// TIA Portal V20 export
FUNCTION "CallCycleTimer" : Void   // FC18, LAD
// stored: SetENOAutomatically false
   VAR CONSTANT
      TRUE : Bool := TRUE;
   END_VAR
BEGIN

REGION Network 1: Cycle Timer Em 0
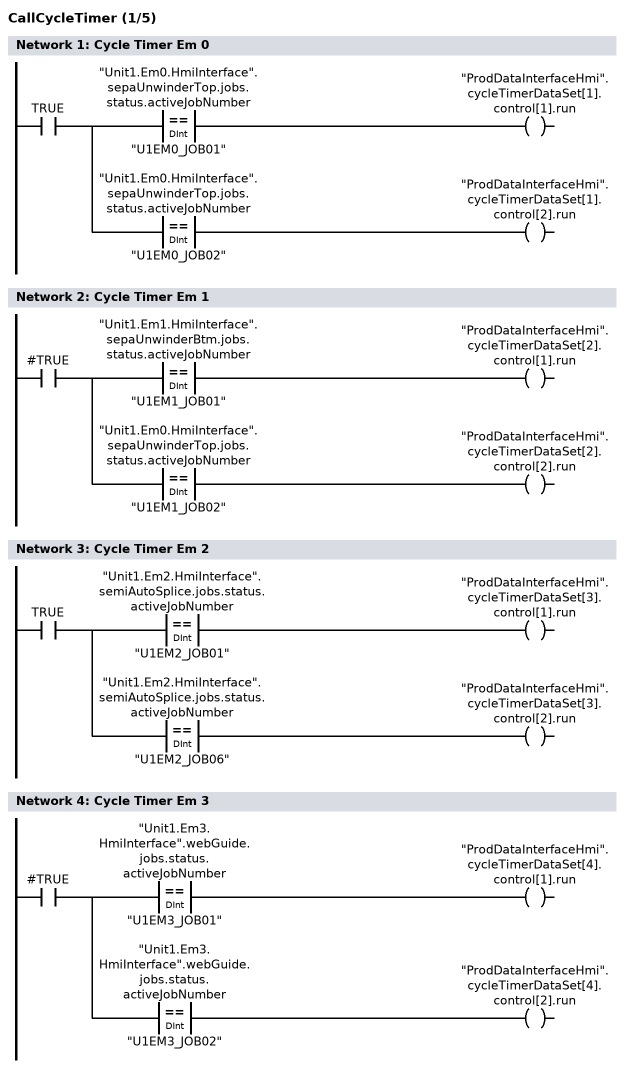
   RUNG wire#powerrail
      Contact( TRUE )
      wire#w1
      { S7_Templates := "SrcType := DInt" } EQ_Contact(in1 := "Unit1.Em0.HmiInterface".sepaUnwinderTop.jobs.status.activeJobNumber, in2 := "U1EM0_JOB01")
      Coil( "ProdDataInterfaceHmi".cycleTimerDataSet[1].control[1].run )
   END_RUNG
   RUNG wire#w1
      { S7_Templates := "SrcType := DInt" } EQ_Contact(in1 := "Unit1.Em0.HmiInterface".sepaUnwinderTop.jobs.status.activeJobNumber, in2 := "U1EM0_JOB02")
      Coil( "ProdDataInterfaceHmi".cycleTimerDataSet[1].control[2].run )
   END_RUNG
   // the same network as SCL:
   "ProdDataInterfaceHmi".cycleTimerDataSet[1].control[1].run := TRUE AND ("Unit1.Em0.HmiInterface".sepaUnwinderTop.jobs.status.activeJobNumber = "U1EM0_JOB01");
   "ProdDataInterfaceHmi".cycleTimerDataSet[1].control[2].run := TRUE AND ("Unit1.Em0.HmiInterface".sepaUnwinderTop.jobs.status.activeJobNumber = "U1EM0_JOB02");
END_REGION

REGION Network 2: Cycle Timer Em 1
   RUNG wire#powerrail
      Contact( #TRUE )
      wire#w1
      { S7_Templates := "SrcType := DInt" } EQ_Contact(in1 := "Unit1.Em1.HmiInterface".sepaUnwinderBtm.jobs.status.activeJobNumber, in2 := "U1EM1_JOB01")
      Coil( "ProdDataInterfaceHmi".cycleTimerDataSet[2].control[1].run )
   END_RUNG
   RUNG wire#w1
      { S7_Templates := "SrcType := DInt" } EQ_Contact(in1 := "Unit1.Em0.HmiInterface".sepaUnwinderTop.jobs.status.activeJobNumber, in2 := "U1EM1_JOB02")
      Coil( "ProdDataInterfaceHmi".cycleTimerDataSet[2].control[2].run )
   END_RUNG
   // the same network as SCL:
   "ProdDataInterfaceHmi".cycleTimerDataSet[2].control[1].run := #TRUE AND ("Unit1.Em1.HmiInterface".sepaUnwinderBtm.jobs.status.activeJobNumber = "U1EM1_JOB01");
   "ProdDataInterfaceHmi".cycleTimerDataSet[2].control[2].run := #TRUE AND ("Unit1.Em0.HmiInterface".sepaUnwinderTop.jobs.status.activeJobNumber = "U1EM1_JOB02");
END_REGION

REGION Network 3: Cycle Timer Em 2
   RUNG wire#powerrail
      Contact( TRUE )
      wire#w1
      { S7_Templates := "SrcType := DInt" } EQ_Contact(in1 := "Unit1.Em2.HmiInterface".semiAutoSplice.jobs.status.activeJobNumber, in2 := "U1EM2_JOB01")
      Coil( "ProdDataInterfaceHmi".cycleTimerDataSet[3].control[1].run )
   END_RUNG
   RUNG wire#w1
      { S7_Templates := "SrcType := DInt" } EQ_Contact(in1 := "Unit1.Em2.HmiInterface".semiAutoSplice.jobs.status.activeJobNumber, in2 := "U1EM2_JOB06")
      Coil( "ProdDataInterfaceHmi".cycleTimerDataSet[3].control[2].run )
   END_RUNG
   // the same network as SCL:
   "ProdDataInterfaceHmi".cycleTimerDataSet[3].control[1].run := TRUE AND ("Unit1.Em2.HmiInterface".semiAutoSplice.jobs.status.activeJobNumber = "U1EM2_JOB01");
   "ProdDataInterfaceHmi".cycleTimerDataSet[3].control[2].run := TRUE AND ("Unit1.Em2.HmiInterface".semiAutoSplice.jobs.status.activeJobNumber = "U1EM2_JOB06");
END_REGION

REGION Network 4: Cycle Timer Em 3
   RUNG wire#powerrail
      Contact( #TRUE )
      wire#w1
      { S7_Templates := "SrcType := DInt" } EQ_Contact(in1 := "Unit1.Em3.HmiInterface".webGuide.jobs.status.activeJobNumber, in2 := "U1EM3_JOB01")
      Coil( "ProdDataInterfaceHmi".cycleTimerDataSet[4].control[1].run )
   END_RUNG
   RUNG wire#w1
      { S7_Templates := "SrcType := DInt" } EQ_Contact(in1 := "Unit1.Em3.HmiInterface".webGuide.jobs.status.activeJobNumber, in2 := "U1EM3_JOB02")
      Coil( "ProdDataInterfaceHmi".cycleTimerDataSet[4].control[2].run )
   END_RUNG
   // the same network as SCL:
   "ProdDataInterfaceHmi".cycleTimerDataSet[4].control[1].run := #TRUE AND ("Unit1.Em3.HmiInterface".webGuide.jobs.status.activeJobNumber = "U1EM3_JOB01");
   "ProdDataInterfaceHmi".cycleTimerDataSet[4].control[2].run := #TRUE AND ("Unit1.Em3.HmiInterface".webGuide.jobs.status.activeJobNumber = "U1EM3_JOB02");
END_REGION

REGION Network 5: Cycle Timer Em 4
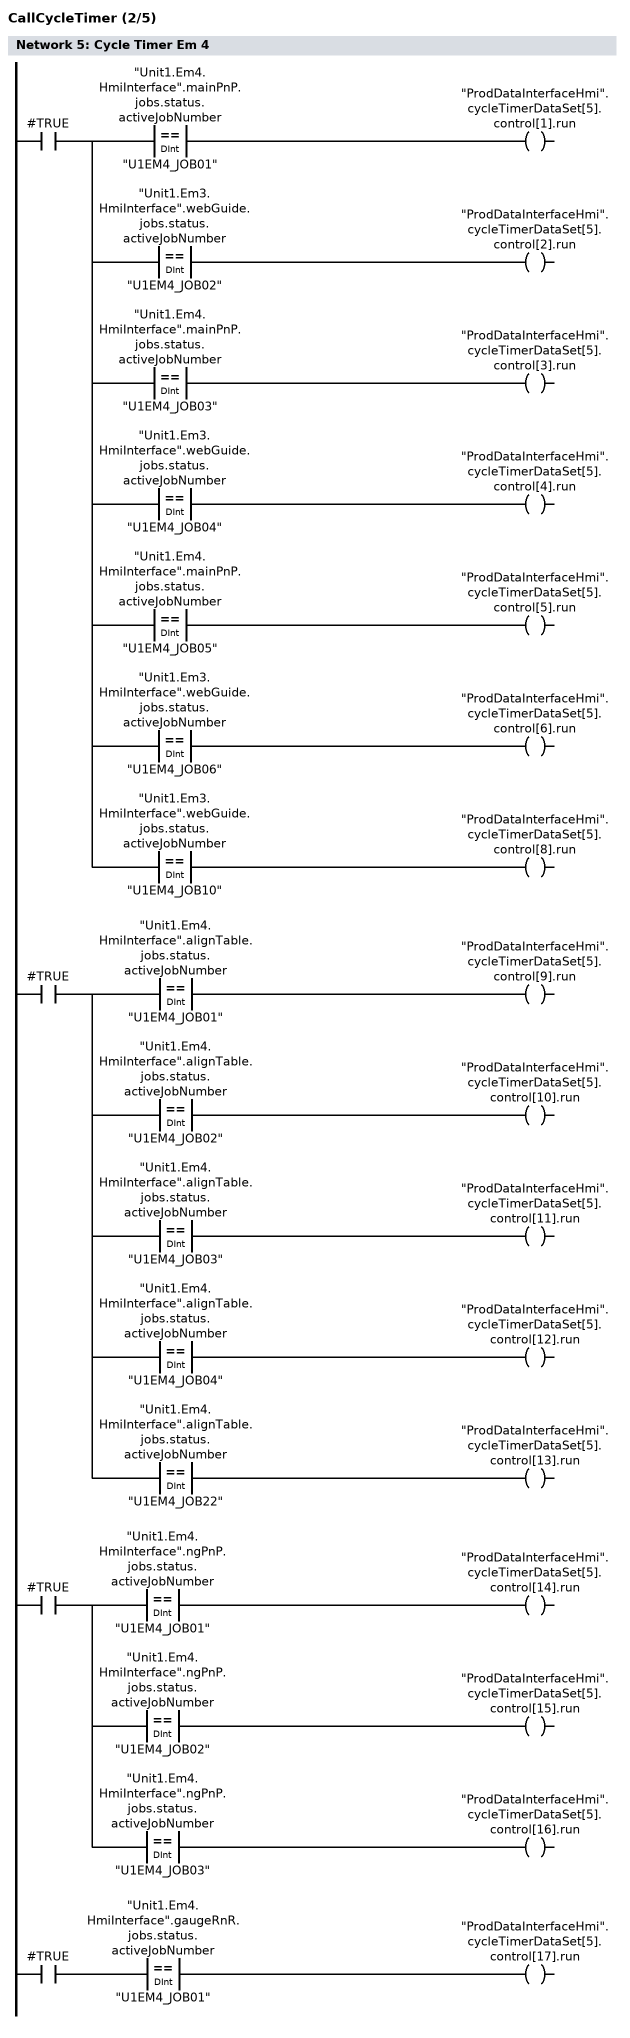
   RUNG wire#powerrail
      Contact( #TRUE )
      wire#w1
      { S7_Templates := "SrcType := DInt" } EQ_Contact(in1 := "Unit1.Em4.HmiInterface".mainPnP.jobs.status.activeJobNumber, in2 := "U1EM4_JOB01")
      Coil( "ProdDataInterfaceHmi".cycleTimerDataSet[5].control[1].run )
   END_RUNG
   RUNG wire#w1
      { S7_Templates := "SrcType := DInt" } EQ_Contact(in1 := "Unit1.Em3.HmiInterface".webGuide.jobs.status.activeJobNumber, in2 := "U1EM4_JOB02")
      Coil( "ProdDataInterfaceHmi".cycleTimerDataSet[5].control[2].run )
   END_RUNG
   RUNG wire#w1
      { S7_Templates := "SrcType := DInt" } EQ_Contact(in1 := "Unit1.Em4.HmiInterface".mainPnP.jobs.status.activeJobNumber, in2 := "U1EM4_JOB03")
      Coil( "ProdDataInterfaceHmi".cycleTimerDataSet[5].control[3].run )
   END_RUNG
   RUNG wire#w1
      { S7_Templates := "SrcType := DInt" } EQ_Contact(in1 := "Unit1.Em3.HmiInterface".webGuide.jobs.status.activeJobNumber, in2 := "U1EM4_JOB04")
      Coil( "ProdDataInterfaceHmi".cycleTimerDataSet[5].control[4].run )
   END_RUNG
   RUNG wire#w1
      { S7_Templates := "SrcType := DInt" } EQ_Contact(in1 := "Unit1.Em4.HmiInterface".mainPnP.jobs.status.activeJobNumber, in2 := "U1EM4_JOB05")
      Coil( "ProdDataInterfaceHmi".cycleTimerDataSet[5].control[5].run )
   END_RUNG
   RUNG wire#w1
      { S7_Templates := "SrcType := DInt" } EQ_Contact(in1 := "Unit1.Em3.HmiInterface".webGuide.jobs.status.activeJobNumber, in2 := "U1EM4_JOB06")
      Coil( "ProdDataInterfaceHmi".cycleTimerDataSet[5].control[6].run )
   END_RUNG
   RUNG wire#w1
      { S7_Templates := "SrcType := DInt" } EQ_Contact(in1 := "Unit1.Em3.HmiInterface".webGuide.jobs.status.activeJobNumber, in2 := "U1EM4_JOB10")
      Coil( "ProdDataInterfaceHmi".cycleTimerDataSet[5].control[8].run )
   END_RUNG
   RUNG wire#powerrail
      Contact( #TRUE )
      wire#w2
      { S7_Templates := "SrcType := DInt" } EQ_Contact(in1 := "Unit1.Em4.HmiInterface".alignTable.jobs.status.activeJobNumber, in2 := "U1EM4_JOB01")
      Coil( "ProdDataInterfaceHmi".cycleTimerDataSet[5].control[9].run )
   END_RUNG
   RUNG wire#w2
      { S7_Templates := "SrcType := DInt" } EQ_Contact(in1 := "Unit1.Em4.HmiInterface".alignTable.jobs.status.activeJobNumber, in2 := "U1EM4_JOB02")
      Coil( "ProdDataInterfaceHmi".cycleTimerDataSet[5].control[10].run )
   END_RUNG
   RUNG wire#w2
      { S7_Templates := "SrcType := DInt" } EQ_Contact(in1 := "Unit1.Em4.HmiInterface".alignTable.jobs.status.activeJobNumber, in2 := "U1EM4_JOB03")
      Coil( "ProdDataInterfaceHmi".cycleTimerDataSet[5].control[11].run )
   END_RUNG
   RUNG wire#w2
      { S7_Templates := "SrcType := DInt" } EQ_Contact(in1 := "Unit1.Em4.HmiInterface".alignTable.jobs.status.activeJobNumber, in2 := "U1EM4_JOB04")
      Coil( "ProdDataInterfaceHmi".cycleTimerDataSet[5].control[12].run )
   END_RUNG
   RUNG wire#w2
      { S7_Templates := "SrcType := DInt" } EQ_Contact(in1 := "Unit1.Em4.HmiInterface".alignTable.jobs.status.activeJobNumber, in2 := "U1EM4_JOB22")
      Coil( "ProdDataInterfaceHmi".cycleTimerDataSet[5].control[13].run )
   END_RUNG
   RUNG wire#powerrail
      Contact( #TRUE )
      wire#w3
      { S7_Templates := "SrcType := DInt" } EQ_Contact(in1 := "Unit1.Em4.HmiInterface".ngPnP.jobs.status.activeJobNumber, in2 := "U1EM4_JOB01")
      Coil( "ProdDataInterfaceHmi".cycleTimerDataSet[5].control[14].run )
   END_RUNG
   RUNG wire#w3
      { S7_Templates := "SrcType := DInt" } EQ_Contact(in1 := "Unit1.Em4.HmiInterface".ngPnP.jobs.status.activeJobNumber, in2 := "U1EM4_JOB02")
      Coil( "ProdDataInterfaceHmi".cycleTimerDataSet[5].control[15].run )
   END_RUNG
   RUNG wire#w3
      { S7_Templates := "SrcType := DInt" } EQ_Contact(in1 := "Unit1.Em4.HmiInterface".ngPnP.jobs.status.activeJobNumber, in2 := "U1EM4_JOB03")
      Coil( "ProdDataInterfaceHmi".cycleTimerDataSet[5].control[16].run )
   END_RUNG
   RUNG wire#powerrail
      Contact( #TRUE )
      { S7_Templates := "SrcType := DInt" } EQ_Contact(in1 := "Unit1.Em4.HmiInterface".gaugeRnR.jobs.status.activeJobNumber, in2 := "U1EM4_JOB01")
      Coil( "ProdDataInterfaceHmi".cycleTimerDataSet[5].control[17].run )
   END_RUNG
   // the same network as SCL:
   "ProdDataInterfaceHmi".cycleTimerDataSet[5].control[1].run := #TRUE AND ("Unit1.Em4.HmiInterface".mainPnP.jobs.status.activeJobNumber = "U1EM4_JOB01");
   "ProdDataInterfaceHmi".cycleTimerDataSet[5].control[2].run := #TRUE AND ("Unit1.Em3.HmiInterface".webGuide.jobs.status.activeJobNumber = "U1EM4_JOB02");
   "ProdDataInterfaceHmi".cycleTimerDataSet[5].control[3].run := #TRUE AND ("Unit1.Em4.HmiInterface".mainPnP.jobs.status.activeJobNumber = "U1EM4_JOB03");
   "ProdDataInterfaceHmi".cycleTimerDataSet[5].control[4].run := #TRUE AND ("Unit1.Em3.HmiInterface".webGuide.jobs.status.activeJobNumber = "U1EM4_JOB04");
   "ProdDataInterfaceHmi".cycleTimerDataSet[5].control[5].run := #TRUE AND ("Unit1.Em4.HmiInterface".mainPnP.jobs.status.activeJobNumber = "U1EM4_JOB05");
   "ProdDataInterfaceHmi".cycleTimerDataSet[5].control[6].run := #TRUE AND ("Unit1.Em3.HmiInterface".webGuide.jobs.status.activeJobNumber = "U1EM4_JOB06");
   "ProdDataInterfaceHmi".cycleTimerDataSet[5].control[8].run := #TRUE AND ("Unit1.Em3.HmiInterface".webGuide.jobs.status.activeJobNumber = "U1EM4_JOB10");
   "ProdDataInterfaceHmi".cycleTimerDataSet[5].control[9].run := #TRUE AND ("Unit1.Em4.HmiInterface".alignTable.jobs.status.activeJobNumber = "U1EM4_JOB01");
   "ProdDataInterfaceHmi".cycleTimerDataSet[5].control[10].run := #TRUE AND ("Unit1.Em4.HmiInterface".alignTable.jobs.status.activeJobNumber = "U1EM4_JOB02");
   "ProdDataInterfaceHmi".cycleTimerDataSet[5].control[11].run := #TRUE AND ("Unit1.Em4.HmiInterface".alignTable.jobs.status.activeJobNumber = "U1EM4_JOB03");
   "ProdDataInterfaceHmi".cycleTimerDataSet[5].control[12].run := #TRUE AND ("Unit1.Em4.HmiInterface".alignTable.jobs.status.activeJobNumber = "U1EM4_JOB04");
   "ProdDataInterfaceHmi".cycleTimerDataSet[5].control[13].run := #TRUE AND ("Unit1.Em4.HmiInterface".alignTable.jobs.status.activeJobNumber = "U1EM4_JOB22");
   "ProdDataInterfaceHmi".cycleTimerDataSet[5].control[14].run := #TRUE AND ("Unit1.Em4.HmiInterface".ngPnP.jobs.status.activeJobNumber = "U1EM4_JOB01");
   "ProdDataInterfaceHmi".cycleTimerDataSet[5].control[15].run := #TRUE AND ("Unit1.Em4.HmiInterface".ngPnP.jobs.status.activeJobNumber = "U1EM4_JOB02");
   "ProdDataInterfaceHmi".cycleTimerDataSet[5].control[16].run := #TRUE AND ("Unit1.Em4.HmiInterface".ngPnP.jobs.status.activeJobNumber = "U1EM4_JOB03");
   "ProdDataInterfaceHmi".cycleTimerDataSet[5].control[17].run := #TRUE AND ("Unit1.Em4.HmiInterface".gaugeRnR.jobs.status.activeJobNumber = "U1EM4_JOB01");
END_REGION

REGION Network 6: Cycle Timer Em 5
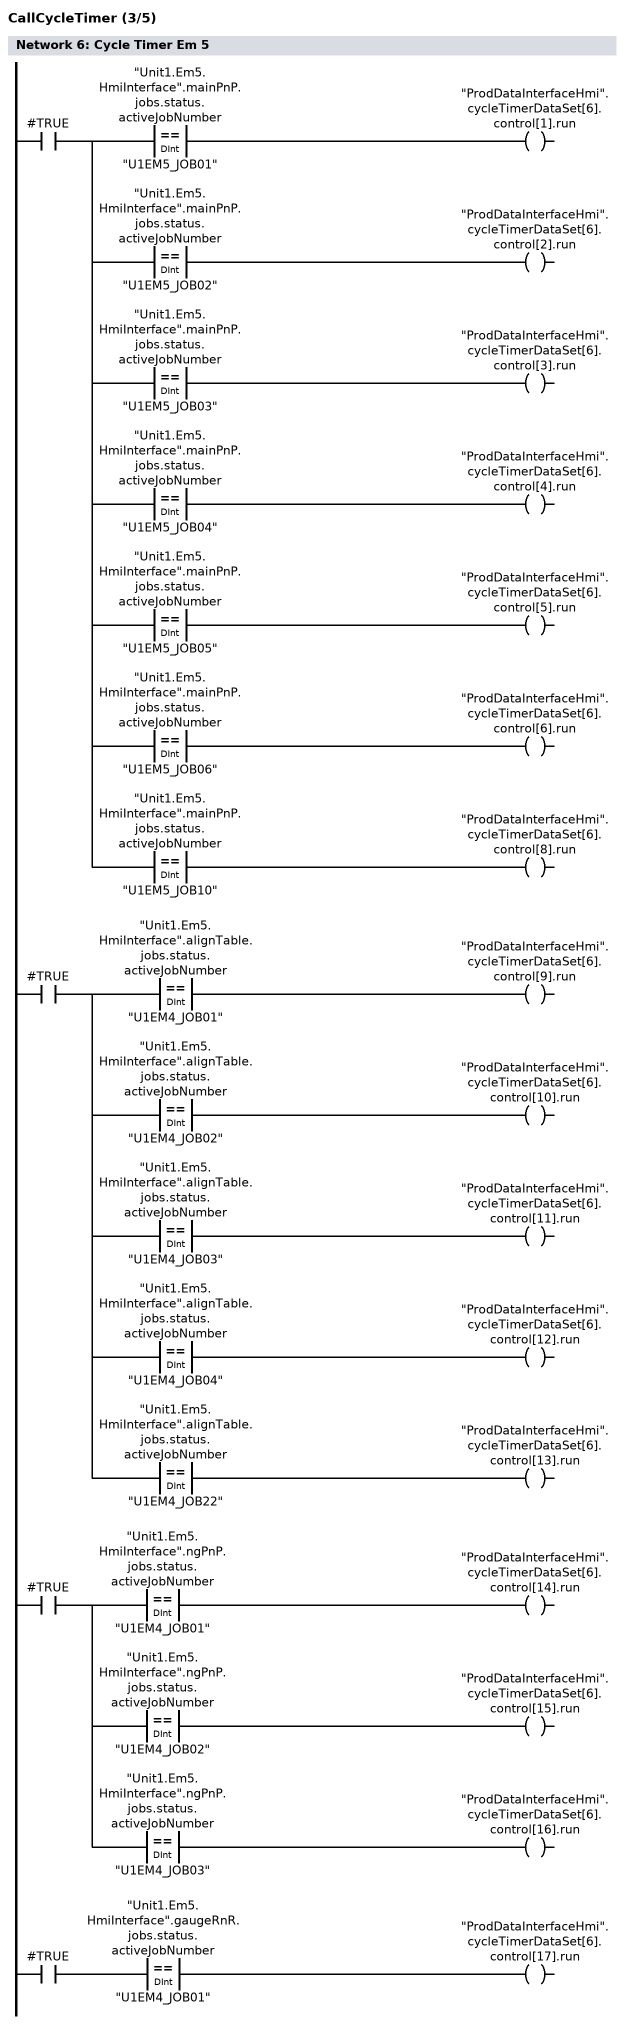
   RUNG wire#powerrail
      Contact( #TRUE )
      wire#w1
      { S7_Templates := "SrcType := DInt" } EQ_Contact(in1 := "Unit1.Em5.HmiInterface".mainPnP.jobs.status.activeJobNumber, in2 := "U1EM5_JOB01")
      Coil( "ProdDataInterfaceHmi".cycleTimerDataSet[6].control[1].run )
   END_RUNG
   RUNG wire#w1
      { S7_Templates := "SrcType := DInt" } EQ_Contact(in1 := "Unit1.Em5.HmiInterface".mainPnP.jobs.status.activeJobNumber, in2 := "U1EM5_JOB02")
      Coil( "ProdDataInterfaceHmi".cycleTimerDataSet[6].control[2].run )
   END_RUNG
   RUNG wire#w1
      { S7_Templates := "SrcType := DInt" } EQ_Contact(in1 := "Unit1.Em5.HmiInterface".mainPnP.jobs.status.activeJobNumber, in2 := "U1EM5_JOB03")
      Coil( "ProdDataInterfaceHmi".cycleTimerDataSet[6].control[3].run )
   END_RUNG
   RUNG wire#w1
      { S7_Templates := "SrcType := DInt" } EQ_Contact(in1 := "Unit1.Em5.HmiInterface".mainPnP.jobs.status.activeJobNumber, in2 := "U1EM5_JOB04")
      Coil( "ProdDataInterfaceHmi".cycleTimerDataSet[6].control[4].run )
   END_RUNG
   RUNG wire#w1
      { S7_Templates := "SrcType := DInt" } EQ_Contact(in1 := "Unit1.Em5.HmiInterface".mainPnP.jobs.status.activeJobNumber, in2 := "U1EM5_JOB05")
      Coil( "ProdDataInterfaceHmi".cycleTimerDataSet[6].control[5].run )
   END_RUNG
   RUNG wire#w1
      { S7_Templates := "SrcType := DInt" } EQ_Contact(in1 := "Unit1.Em5.HmiInterface".mainPnP.jobs.status.activeJobNumber, in2 := "U1EM5_JOB06")
      Coil( "ProdDataInterfaceHmi".cycleTimerDataSet[6].control[6].run )
   END_RUNG
   RUNG wire#w1
      { S7_Templates := "SrcType := DInt" } EQ_Contact(in1 := "Unit1.Em5.HmiInterface".mainPnP.jobs.status.activeJobNumber, in2 := "U1EM5_JOB10")
      Coil( "ProdDataInterfaceHmi".cycleTimerDataSet[6].control[8].run )
   END_RUNG
   RUNG wire#powerrail
      Contact( #TRUE )
      wire#w2
      { S7_Templates := "SrcType := DInt" } EQ_Contact(in1 := "Unit1.Em5.HmiInterface".alignTable.jobs.status.activeJobNumber, in2 := "U1EM4_JOB01")
      Coil( "ProdDataInterfaceHmi".cycleTimerDataSet[6].control[9].run )
   END_RUNG
   RUNG wire#w2
      { S7_Templates := "SrcType := DInt" } EQ_Contact(in1 := "Unit1.Em5.HmiInterface".alignTable.jobs.status.activeJobNumber, in2 := "U1EM4_JOB02")
      Coil( "ProdDataInterfaceHmi".cycleTimerDataSet[6].control[10].run )
   END_RUNG
   RUNG wire#w2
      { S7_Templates := "SrcType := DInt" } EQ_Contact(in1 := "Unit1.Em5.HmiInterface".alignTable.jobs.status.activeJobNumber, in2 := "U1EM4_JOB03")
      Coil( "ProdDataInterfaceHmi".cycleTimerDataSet[6].control[11].run )
   END_RUNG
   RUNG wire#w2
      { S7_Templates := "SrcType := DInt" } EQ_Contact(in1 := "Unit1.Em5.HmiInterface".alignTable.jobs.status.activeJobNumber, in2 := "U1EM4_JOB04")
      Coil( "ProdDataInterfaceHmi".cycleTimerDataSet[6].control[12].run )
   END_RUNG
   RUNG wire#w2
      { S7_Templates := "SrcType := DInt" } EQ_Contact(in1 := "Unit1.Em5.HmiInterface".alignTable.jobs.status.activeJobNumber, in2 := "U1EM4_JOB22")
      Coil( "ProdDataInterfaceHmi".cycleTimerDataSet[6].control[13].run )
   END_RUNG
   RUNG wire#powerrail
      Contact( #TRUE )
      wire#w3
      { S7_Templates := "SrcType := DInt" } EQ_Contact(in1 := "Unit1.Em5.HmiInterface".ngPnP.jobs.status.activeJobNumber, in2 := "U1EM4_JOB01")
      Coil( "ProdDataInterfaceHmi".cycleTimerDataSet[6].control[14].run )
   END_RUNG
   RUNG wire#w3
      { S7_Templates := "SrcType := DInt" } EQ_Contact(in1 := "Unit1.Em5.HmiInterface".ngPnP.jobs.status.activeJobNumber, in2 := "U1EM4_JOB02")
      Coil( "ProdDataInterfaceHmi".cycleTimerDataSet[6].control[15].run )
   END_RUNG
   RUNG wire#w3
      { S7_Templates := "SrcType := DInt" } EQ_Contact(in1 := "Unit1.Em5.HmiInterface".ngPnP.jobs.status.activeJobNumber, in2 := "U1EM4_JOB03")
      Coil( "ProdDataInterfaceHmi".cycleTimerDataSet[6].control[16].run )
   END_RUNG
   RUNG wire#powerrail
      Contact( #TRUE )
      { S7_Templates := "SrcType := DInt" } EQ_Contact(in1 := "Unit1.Em5.HmiInterface".gaugeRnR.jobs.status.activeJobNumber, in2 := "U1EM4_JOB01")
      Coil( "ProdDataInterfaceHmi".cycleTimerDataSet[6].control[17].run )
   END_RUNG
   // the same network as SCL:
   "ProdDataInterfaceHmi".cycleTimerDataSet[6].control[1].run := #TRUE AND ("Unit1.Em5.HmiInterface".mainPnP.jobs.status.activeJobNumber = "U1EM5_JOB01");
   "ProdDataInterfaceHmi".cycleTimerDataSet[6].control[2].run := #TRUE AND ("Unit1.Em5.HmiInterface".mainPnP.jobs.status.activeJobNumber = "U1EM5_JOB02");
   "ProdDataInterfaceHmi".cycleTimerDataSet[6].control[3].run := #TRUE AND ("Unit1.Em5.HmiInterface".mainPnP.jobs.status.activeJobNumber = "U1EM5_JOB03");
   "ProdDataInterfaceHmi".cycleTimerDataSet[6].control[4].run := #TRUE AND ("Unit1.Em5.HmiInterface".mainPnP.jobs.status.activeJobNumber = "U1EM5_JOB04");
   "ProdDataInterfaceHmi".cycleTimerDataSet[6].control[5].run := #TRUE AND ("Unit1.Em5.HmiInterface".mainPnP.jobs.status.activeJobNumber = "U1EM5_JOB05");
   "ProdDataInterfaceHmi".cycleTimerDataSet[6].control[6].run := #TRUE AND ("Unit1.Em5.HmiInterface".mainPnP.jobs.status.activeJobNumber = "U1EM5_JOB06");
   "ProdDataInterfaceHmi".cycleTimerDataSet[6].control[8].run := #TRUE AND ("Unit1.Em5.HmiInterface".mainPnP.jobs.status.activeJobNumber = "U1EM5_JOB10");
   "ProdDataInterfaceHmi".cycleTimerDataSet[6].control[9].run := #TRUE AND ("Unit1.Em5.HmiInterface".alignTable.jobs.status.activeJobNumber = "U1EM4_JOB01");
   "ProdDataInterfaceHmi".cycleTimerDataSet[6].control[10].run := #TRUE AND ("Unit1.Em5.HmiInterface".alignTable.jobs.status.activeJobNumber = "U1EM4_JOB02");
   "ProdDataInterfaceHmi".cycleTimerDataSet[6].control[11].run := #TRUE AND ("Unit1.Em5.HmiInterface".alignTable.jobs.status.activeJobNumber = "U1EM4_JOB03");
   "ProdDataInterfaceHmi".cycleTimerDataSet[6].control[12].run := #TRUE AND ("Unit1.Em5.HmiInterface".alignTable.jobs.status.activeJobNumber = "U1EM4_JOB04");
   "ProdDataInterfaceHmi".cycleTimerDataSet[6].control[13].run := #TRUE AND ("Unit1.Em5.HmiInterface".alignTable.jobs.status.activeJobNumber = "U1EM4_JOB22");
   "ProdDataInterfaceHmi".cycleTimerDataSet[6].control[14].run := #TRUE AND ("Unit1.Em5.HmiInterface".ngPnP.jobs.status.activeJobNumber = "U1EM4_JOB01");
   "ProdDataInterfaceHmi".cycleTimerDataSet[6].control[15].run := #TRUE AND ("Unit1.Em5.HmiInterface".ngPnP.jobs.status.activeJobNumber = "U1EM4_JOB02");
   "ProdDataInterfaceHmi".cycleTimerDataSet[6].control[16].run := #TRUE AND ("Unit1.Em5.HmiInterface".ngPnP.jobs.status.activeJobNumber = "U1EM4_JOB03");
   "ProdDataInterfaceHmi".cycleTimerDataSet[6].control[17].run := #TRUE AND ("Unit1.Em5.HmiInterface".gaugeRnR.jobs.status.activeJobNumber = "U1EM4_JOB01");
END_REGION

REGION Network 7: Cycle Timer Em 6
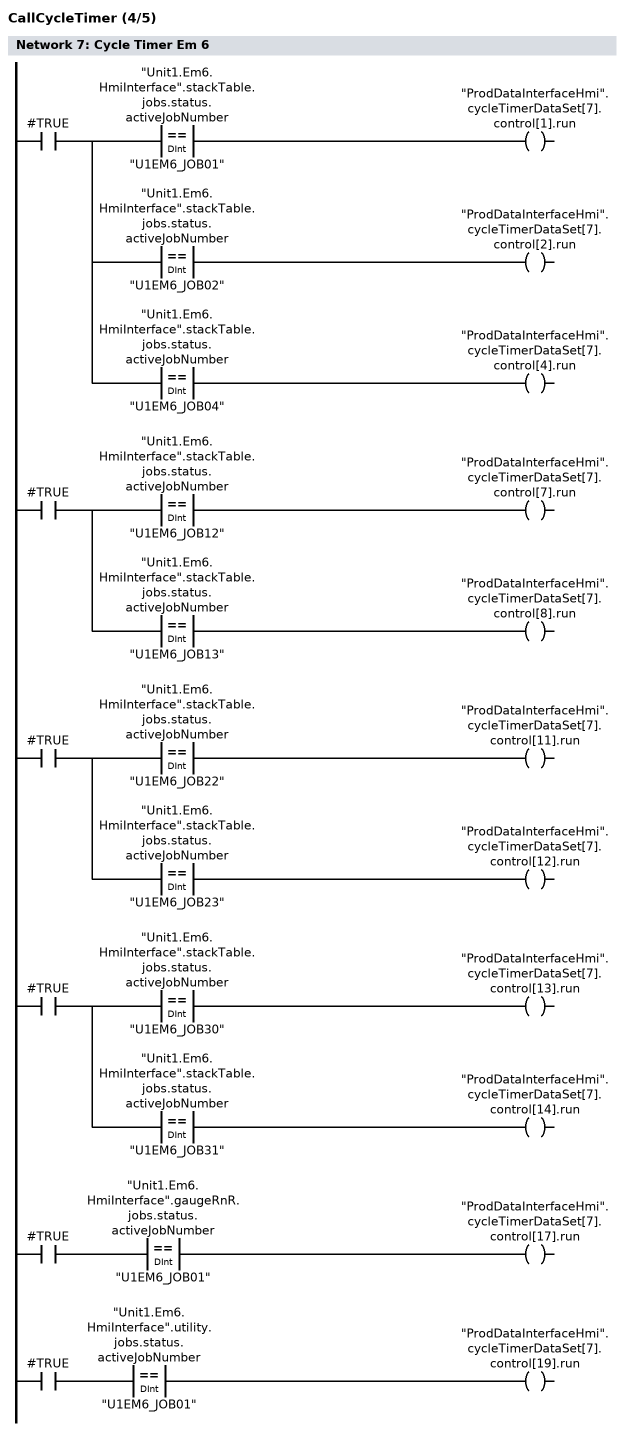
   RUNG wire#powerrail
      Contact( #TRUE )
      wire#w1
      { S7_Templates := "SrcType := DInt" } EQ_Contact(in1 := "Unit1.Em6.HmiInterface".stackTable.jobs.status.activeJobNumber, in2 := "U1EM6_JOB01")
      Coil( "ProdDataInterfaceHmi".cycleTimerDataSet[7].control[1].run )
   END_RUNG
   RUNG wire#w1
      { S7_Templates := "SrcType := DInt" } EQ_Contact(in1 := "Unit1.Em6.HmiInterface".stackTable.jobs.status.activeJobNumber, in2 := "U1EM6_JOB02")
      Coil( "ProdDataInterfaceHmi".cycleTimerDataSet[7].control[2].run )
   END_RUNG
   RUNG wire#w1
      { S7_Templates := "SrcType := DInt" } EQ_Contact(in1 := "Unit1.Em6.HmiInterface".stackTable.jobs.status.activeJobNumber, in2 := "U1EM6_JOB04")
      Coil( "ProdDataInterfaceHmi".cycleTimerDataSet[7].control[4].run )
   END_RUNG
   RUNG wire#powerrail
      Contact( #TRUE )
      wire#w2
      { S7_Templates := "SrcType := DInt" } EQ_Contact(in1 := "Unit1.Em6.HmiInterface".stackTable.jobs.status.activeJobNumber, in2 := "U1EM6_JOB12")
      Coil( "ProdDataInterfaceHmi".cycleTimerDataSet[7].control[7].run )
   END_RUNG
   RUNG wire#w2
      { S7_Templates := "SrcType := DInt" } EQ_Contact(in1 := "Unit1.Em6.HmiInterface".stackTable.jobs.status.activeJobNumber, in2 := "U1EM6_JOB13")
      Coil( "ProdDataInterfaceHmi".cycleTimerDataSet[7].control[8].run )
   END_RUNG
   RUNG wire#powerrail
      Contact( #TRUE )
      wire#w3
      { S7_Templates := "SrcType := DInt" } EQ_Contact(in1 := "Unit1.Em6.HmiInterface".stackTable.jobs.status.activeJobNumber, in2 := "U1EM6_JOB22")
      Coil( "ProdDataInterfaceHmi".cycleTimerDataSet[7].control[11].run )
   END_RUNG
   RUNG wire#w3
      { S7_Templates := "SrcType := DInt" } EQ_Contact(in1 := "Unit1.Em6.HmiInterface".stackTable.jobs.status.activeJobNumber, in2 := "U1EM6_JOB23")
      Coil( "ProdDataInterfaceHmi".cycleTimerDataSet[7].control[12].run )
   END_RUNG
   RUNG wire#powerrail
      Contact( #TRUE )
      wire#w4
      { S7_Templates := "SrcType := DInt" } EQ_Contact(in1 := "Unit1.Em6.HmiInterface".stackTable.jobs.status.activeJobNumber, in2 := "U1EM6_JOB30")
      Coil( "ProdDataInterfaceHmi".cycleTimerDataSet[7].control[13].run )
   END_RUNG
   RUNG wire#w4
      { S7_Templates := "SrcType := DInt" } EQ_Contact(in1 := "Unit1.Em6.HmiInterface".stackTable.jobs.status.activeJobNumber, in2 := "U1EM6_JOB31")
      Coil( "ProdDataInterfaceHmi".cycleTimerDataSet[7].control[14].run )
   END_RUNG
   RUNG wire#powerrail
      Contact( #TRUE )
      { S7_Templates := "SrcType := DInt" } EQ_Contact(in1 := "Unit1.Em6.HmiInterface".gaugeRnR.jobs.status.activeJobNumber, in2 := "U1EM6_JOB01")
      Coil( "ProdDataInterfaceHmi".cycleTimerDataSet[7].control[17].run )
   END_RUNG
   RUNG wire#powerrail
      Contact( #TRUE )
      { S7_Templates := "SrcType := DInt" } EQ_Contact(in1 := "Unit1.Em6.HmiInterface".utility.jobs.status.activeJobNumber, in2 := "U1EM6_JOB01")
      Coil( "ProdDataInterfaceHmi".cycleTimerDataSet[7].control[19].run )
   END_RUNG
   // the same network as SCL:
   "ProdDataInterfaceHmi".cycleTimerDataSet[7].control[1].run := #TRUE AND ("Unit1.Em6.HmiInterface".stackTable.jobs.status.activeJobNumber = "U1EM6_JOB01");
   "ProdDataInterfaceHmi".cycleTimerDataSet[7].control[2].run := #TRUE AND ("Unit1.Em6.HmiInterface".stackTable.jobs.status.activeJobNumber = "U1EM6_JOB02");
   "ProdDataInterfaceHmi".cycleTimerDataSet[7].control[4].run := #TRUE AND ("Unit1.Em6.HmiInterface".stackTable.jobs.status.activeJobNumber = "U1EM6_JOB04");
   "ProdDataInterfaceHmi".cycleTimerDataSet[7].control[7].run := #TRUE AND ("Unit1.Em6.HmiInterface".stackTable.jobs.status.activeJobNumber = "U1EM6_JOB12");
   "ProdDataInterfaceHmi".cycleTimerDataSet[7].control[8].run := #TRUE AND ("Unit1.Em6.HmiInterface".stackTable.jobs.status.activeJobNumber = "U1EM6_JOB13");
   "ProdDataInterfaceHmi".cycleTimerDataSet[7].control[11].run := #TRUE AND ("Unit1.Em6.HmiInterface".stackTable.jobs.status.activeJobNumber = "U1EM6_JOB22");
   "ProdDataInterfaceHmi".cycleTimerDataSet[7].control[12].run := #TRUE AND ("Unit1.Em6.HmiInterface".stackTable.jobs.status.activeJobNumber = "U1EM6_JOB23");
   "ProdDataInterfaceHmi".cycleTimerDataSet[7].control[13].run := #TRUE AND ("Unit1.Em6.HmiInterface".stackTable.jobs.status.activeJobNumber = "U1EM6_JOB30");
   "ProdDataInterfaceHmi".cycleTimerDataSet[7].control[14].run := #TRUE AND ("Unit1.Em6.HmiInterface".stackTable.jobs.status.activeJobNumber = "U1EM6_JOB31");
   "ProdDataInterfaceHmi".cycleTimerDataSet[7].control[17].run := #TRUE AND ("Unit1.Em6.HmiInterface".gaugeRnR.jobs.status.activeJobNumber = "U1EM6_JOB01");
   "ProdDataInterfaceHmi".cycleTimerDataSet[7].control[19].run := #TRUE AND ("Unit1.Em6.HmiInterface".utility.jobs.status.activeJobNumber = "U1EM6_JOB01");
END_REGION

REGION Network 8: Cycle Timer Em 7
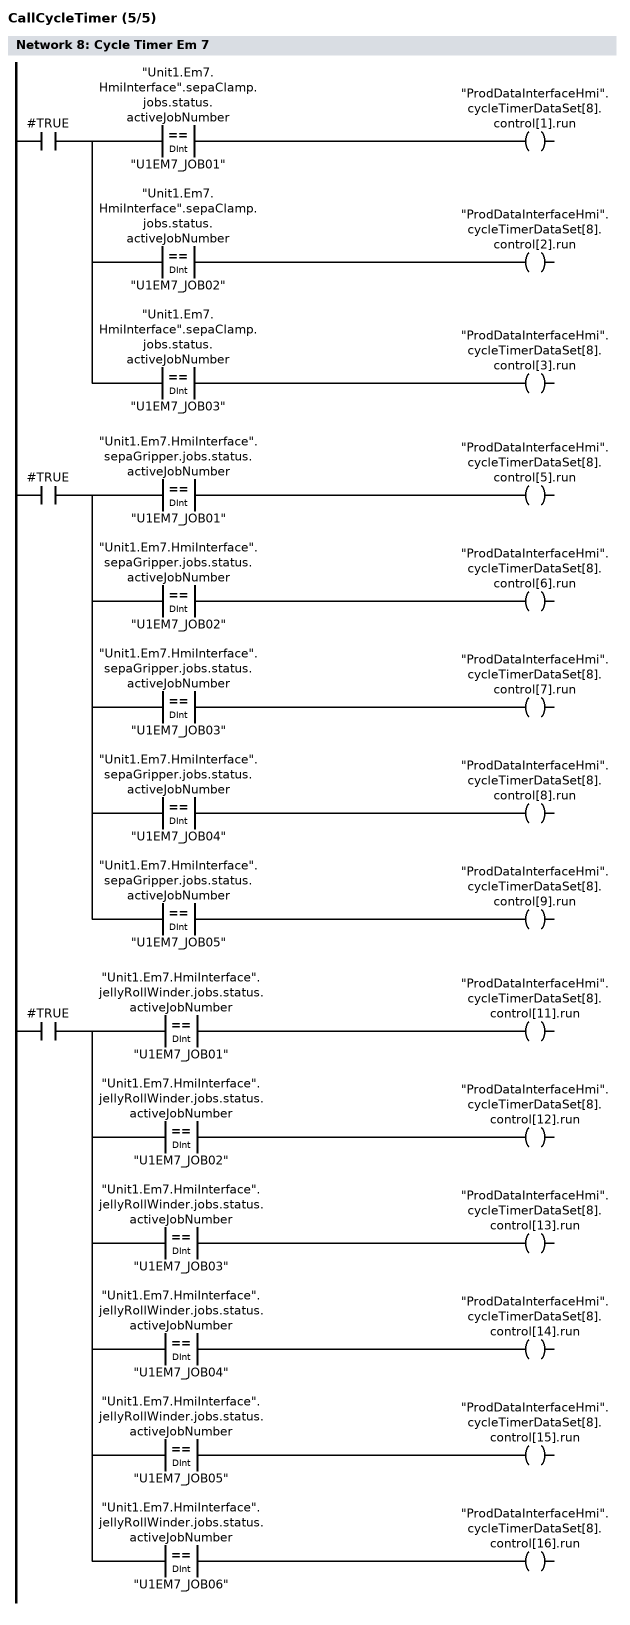
   RUNG wire#powerrail
      Contact( #TRUE )
      wire#w1
      { S7_Templates := "SrcType := DInt" } EQ_Contact(in1 := "Unit1.Em7.HmiInterface".sepaClamp.jobs.status.activeJobNumber, in2 := "U1EM7_JOB01")
      Coil( "ProdDataInterfaceHmi".cycleTimerDataSet[8].control[1].run )
   END_RUNG
   RUNG wire#w1
      { S7_Templates := "SrcType := DInt" } EQ_Contact(in1 := "Unit1.Em7.HmiInterface".sepaClamp.jobs.status.activeJobNumber, in2 := "U1EM7_JOB02")
      Coil( "ProdDataInterfaceHmi".cycleTimerDataSet[8].control[2].run )
   END_RUNG
   RUNG wire#w1
      { S7_Templates := "SrcType := DInt" } EQ_Contact(in1 := "Unit1.Em7.HmiInterface".sepaClamp.jobs.status.activeJobNumber, in2 := "U1EM7_JOB03")
      Coil( "ProdDataInterfaceHmi".cycleTimerDataSet[8].control[3].run )
   END_RUNG
   RUNG wire#powerrail
      Contact( #TRUE )
      wire#w2
      { S7_Templates := "SrcType := DInt" } EQ_Contact(in1 := "Unit1.Em7.HmiInterface".sepaGripper.jobs.status.activeJobNumber, in2 := "U1EM7_JOB01")
      Coil( "ProdDataInterfaceHmi".cycleTimerDataSet[8].control[5].run )
   END_RUNG
   RUNG wire#w2
      { S7_Templates := "SrcType := DInt" } EQ_Contact(in1 := "Unit1.Em7.HmiInterface".sepaGripper.jobs.status.activeJobNumber, in2 := "U1EM7_JOB02")
      Coil( "ProdDataInterfaceHmi".cycleTimerDataSet[8].control[6].run )
   END_RUNG
   RUNG wire#w2
      { S7_Templates := "SrcType := DInt" } EQ_Contact(in1 := "Unit1.Em7.HmiInterface".sepaGripper.jobs.status.activeJobNumber, in2 := "U1EM7_JOB03")
      Coil( "ProdDataInterfaceHmi".cycleTimerDataSet[8].control[7].run )
   END_RUNG
   RUNG wire#w2
      { S7_Templates := "SrcType := DInt" } EQ_Contact(in1 := "Unit1.Em7.HmiInterface".sepaGripper.jobs.status.activeJobNumber, in2 := "U1EM7_JOB04")
      Coil( "ProdDataInterfaceHmi".cycleTimerDataSet[8].control[8].run )
   END_RUNG
   RUNG wire#w2
      { S7_Templates := "SrcType := DInt" } EQ_Contact(in1 := "Unit1.Em7.HmiInterface".sepaGripper.jobs.status.activeJobNumber, in2 := "U1EM7_JOB05")
      Coil( "ProdDataInterfaceHmi".cycleTimerDataSet[8].control[9].run )
   END_RUNG
   RUNG wire#powerrail
      Contact( #TRUE )
      wire#w3
      { S7_Templates := "SrcType := DInt" } EQ_Contact(in1 := "Unit1.Em7.HmiInterface".jellyRollWinder.jobs.status.activeJobNumber, in2 := "U1EM7_JOB01")
      Coil( "ProdDataInterfaceHmi".cycleTimerDataSet[8].control[11].run )
   END_RUNG
   RUNG wire#w3
      { S7_Templates := "SrcType := DInt" } EQ_Contact(in1 := "Unit1.Em7.HmiInterface".jellyRollWinder.jobs.status.activeJobNumber, in2 := "U1EM7_JOB02")
      Coil( "ProdDataInterfaceHmi".cycleTimerDataSet[8].control[12].run )
   END_RUNG
   RUNG wire#w3
      { S7_Templates := "SrcType := DInt" } EQ_Contact(in1 := "Unit1.Em7.HmiInterface".jellyRollWinder.jobs.status.activeJobNumber, in2 := "U1EM7_JOB03")
      Coil( "ProdDataInterfaceHmi".cycleTimerDataSet[8].control[13].run )
   END_RUNG
   RUNG wire#w3
      { S7_Templates := "SrcType := DInt" } EQ_Contact(in1 := "Unit1.Em7.HmiInterface".jellyRollWinder.jobs.status.activeJobNumber, in2 := "U1EM7_JOB04")
      Coil( "ProdDataInterfaceHmi".cycleTimerDataSet[8].control[14].run )
   END_RUNG
   RUNG wire#w3
      { S7_Templates := "SrcType := DInt" } EQ_Contact(in1 := "Unit1.Em7.HmiInterface".jellyRollWinder.jobs.status.activeJobNumber, in2 := "U1EM7_JOB05")
      Coil( "ProdDataInterfaceHmi".cycleTimerDataSet[8].control[15].run )
   END_RUNG
   RUNG wire#w3
      { S7_Templates := "SrcType := DInt" } EQ_Contact(in1 := "Unit1.Em7.HmiInterface".jellyRollWinder.jobs.status.activeJobNumber, in2 := "U1EM7_JOB06")
      Coil( "ProdDataInterfaceHmi".cycleTimerDataSet[8].control[16].run )
   END_RUNG
   // the same network as SCL:
   "ProdDataInterfaceHmi".cycleTimerDataSet[8].control[1].run := #TRUE AND ("Unit1.Em7.HmiInterface".sepaClamp.jobs.status.activeJobNumber = "U1EM7_JOB01");
   "ProdDataInterfaceHmi".cycleTimerDataSet[8].control[2].run := #TRUE AND ("Unit1.Em7.HmiInterface".sepaClamp.jobs.status.activeJobNumber = "U1EM7_JOB02");
   "ProdDataInterfaceHmi".cycleTimerDataSet[8].control[3].run := #TRUE AND ("Unit1.Em7.HmiInterface".sepaClamp.jobs.status.activeJobNumber = "U1EM7_JOB03");
   "ProdDataInterfaceHmi".cycleTimerDataSet[8].control[5].run := #TRUE AND ("Unit1.Em7.HmiInterface".sepaGripper.jobs.status.activeJobNumber = "U1EM7_JOB01");
   "ProdDataInterfaceHmi".cycleTimerDataSet[8].control[6].run := #TRUE AND ("Unit1.Em7.HmiInterface".sepaGripper.jobs.status.activeJobNumber = "U1EM7_JOB02");
   "ProdDataInterfaceHmi".cycleTimerDataSet[8].control[7].run := #TRUE AND ("Unit1.Em7.HmiInterface".sepaGripper.jobs.status.activeJobNumber = "U1EM7_JOB03");
   "ProdDataInterfaceHmi".cycleTimerDataSet[8].control[8].run := #TRUE AND ("Unit1.Em7.HmiInterface".sepaGripper.jobs.status.activeJobNumber = "U1EM7_JOB04");
   "ProdDataInterfaceHmi".cycleTimerDataSet[8].control[9].run := #TRUE AND ("Unit1.Em7.HmiInterface".sepaGripper.jobs.status.activeJobNumber = "U1EM7_JOB05");
   "ProdDataInterfaceHmi".cycleTimerDataSet[8].control[11].run := #TRUE AND ("Unit1.Em7.HmiInterface".jellyRollWinder.jobs.status.activeJobNumber = "U1EM7_JOB01");
   "ProdDataInterfaceHmi".cycleTimerDataSet[8].control[12].run := #TRUE AND ("Unit1.Em7.HmiInterface".jellyRollWinder.jobs.status.activeJobNumber = "U1EM7_JOB02");
   "ProdDataInterfaceHmi".cycleTimerDataSet[8].control[13].run := #TRUE AND ("Unit1.Em7.HmiInterface".jellyRollWinder.jobs.status.activeJobNumber = "U1EM7_JOB03");
   "ProdDataInterfaceHmi".cycleTimerDataSet[8].control[14].run := #TRUE AND ("Unit1.Em7.HmiInterface".jellyRollWinder.jobs.status.activeJobNumber = "U1EM7_JOB04");
   "ProdDataInterfaceHmi".cycleTimerDataSet[8].control[15].run := #TRUE AND ("Unit1.Em7.HmiInterface".jellyRollWinder.jobs.status.activeJobNumber = "U1EM7_JOB05");
   "ProdDataInterfaceHmi".cycleTimerDataSet[8].control[16].run := #TRUE AND ("Unit1.Em7.HmiInterface".jellyRollWinder.jobs.status.activeJobNumber = "U1EM7_JOB06");
END_REGION
END_FUNCTION
